TYPE ST_XBox_Trigger_NC_Options :
STRUCT
	// Inverts the direction of the axis
	bInverted : BOOL := FALSE;
	// Maximum Feedrate
	fMaxOverride : LREAL := 100.0;
	// Struct of parameters for MC_Halt command
	stXBox_NC_Halt_Dynamics : ST_XBox_NC_Halt_Dynamics;
END_STRUCT
END_TYPE

(* stored: Version 1.1.0.1, ProductVersion 3.1.4024.11
   DUT ST_XBox_Trigger_NC_Options: Id {227011e3-3da0-45fe-836e-8de3fdd94553} *)
